(* Logix 5000 project; controller SX_V040001_C001 vendor 1 type 14 code 77 rev 16.23; software revision 16.04; part 24 of 35 *)
(* tags used below, declared in another part *)
   ALL_KINDS : INT[90];
   Basic : INT;
   DRIVE : INT[32];
   DRIVE_INTERVAL : INT[8];
   G_AInput : DINT[8];
   G_DInput : DINT[3];
   G_DOutput : DINT[3];
   Min_Counter : DINT;
   PARAMETER : INT[501];
(* MainProgram, continued *)

ROUTINE OperatingHours   (* ladder *)
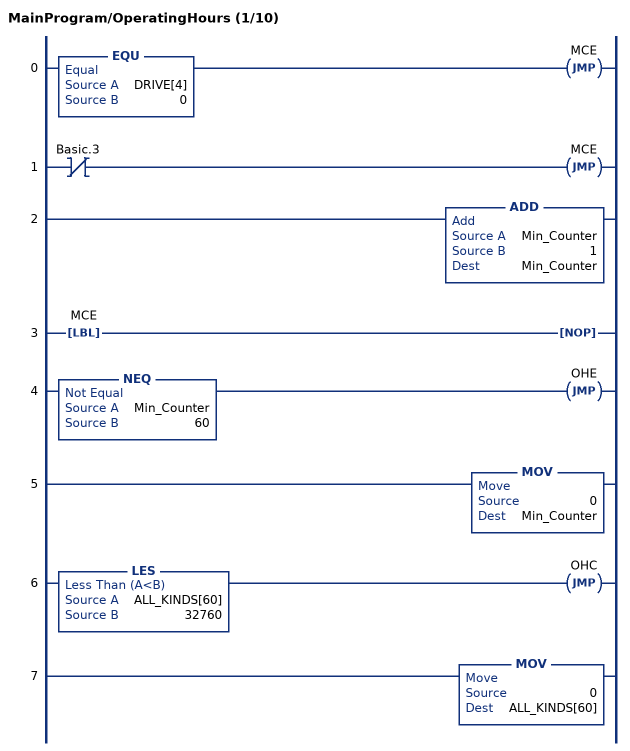
   0: EQU(DRIVE[4],0)JMP(MCE);
   1: XIO(Basic.3)JMP(MCE);
   2: ADD(Min_Counter,1,Min_Counter);
   3: LBL(MCE)NOP();
   4: NEQ(Min_Counter,60)JMP(OHE);
   5: MOV(0,Min_Counter);
   6: LES(ALL_KINDS[60],32760)JMP(OHC);
   7: MOV(0,ALL_KINDS[60]);
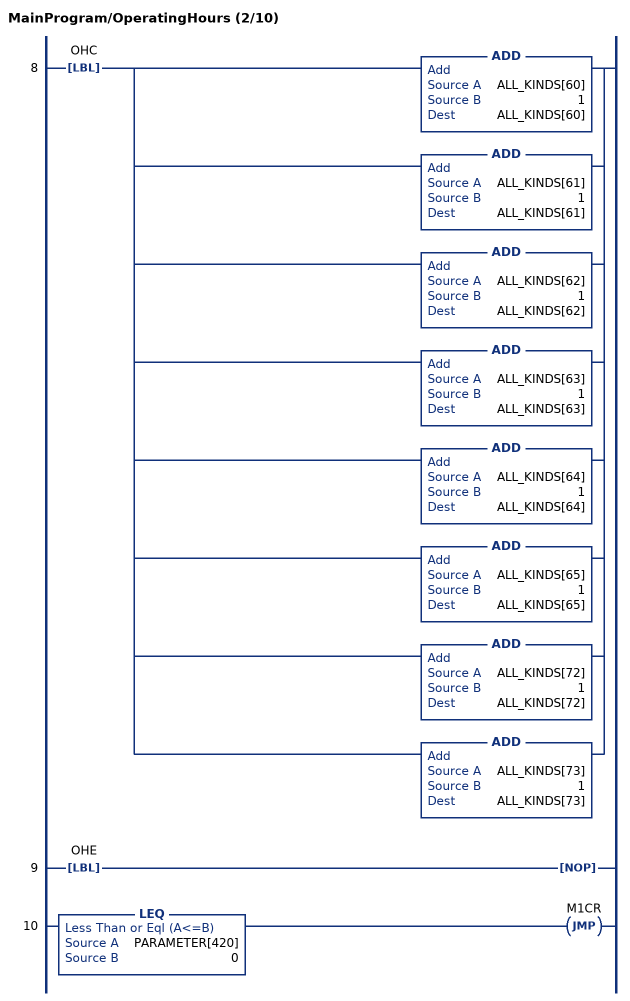
   8: LBL(OHC)[ADD(ALL_KINDS[60],1,ALL_KINDS[60]) ,ADD(ALL_KINDS[61],1,ALL_KINDS[61]) ,ADD(ALL_KINDS[62],1,ALL_KINDS[62]) ,ADD(ALL_KINDS[63],1,ALL_KINDS[63]) ,ADD(ALL_KINDS[64],1,ALL_KINDS[64]) ,ADD(ALL_KINDS[65],1,ALL_KINDS[65]) ,ADD(ALL_KINDS[72],1,ALL_KINDS[72]) ,ADD(ALL_KINDS[73],1,ALL_KINDS[73]) ];
   9: LBL(OHE)NOP();
   10: LEQ(PARAMETER[420],0)JMP(M1CR);
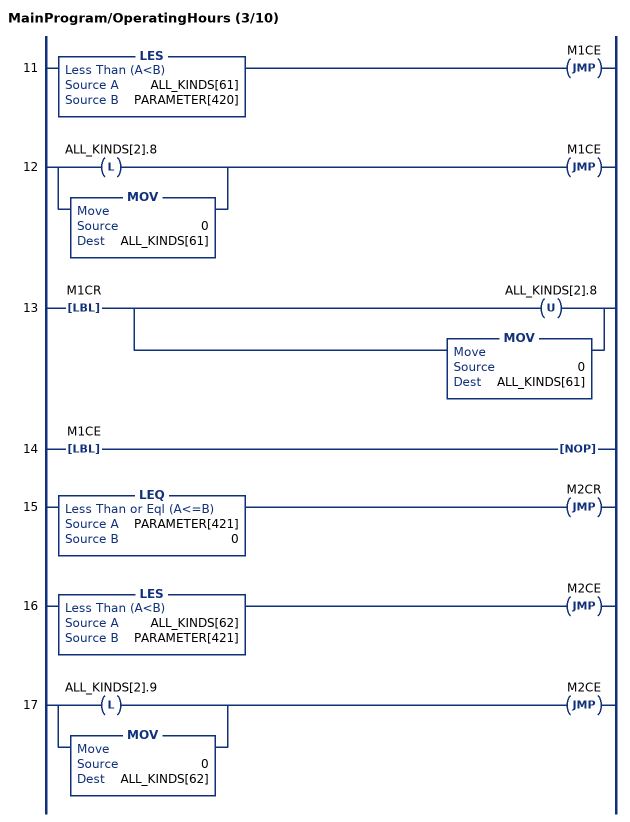
   11: LES(ALL_KINDS[61],PARAMETER[420])JMP(M1CE);
   12: [OTL(ALL_KINDS[2].8) ,MOV(0,ALL_KINDS[61]) ]JMP(M1CE);
   13: LBL(M1CR)[OTU(ALL_KINDS[2].8) ,MOV(0,ALL_KINDS[61]) ];
   14: LBL(M1CE)NOP();
   15: LEQ(PARAMETER[421],0)JMP(M2CR);
   16: LES(ALL_KINDS[62],PARAMETER[421])JMP(M2CE);
   17: [OTL(ALL_KINDS[2].9) ,MOV(0,ALL_KINDS[62]) ]JMP(M2CE);
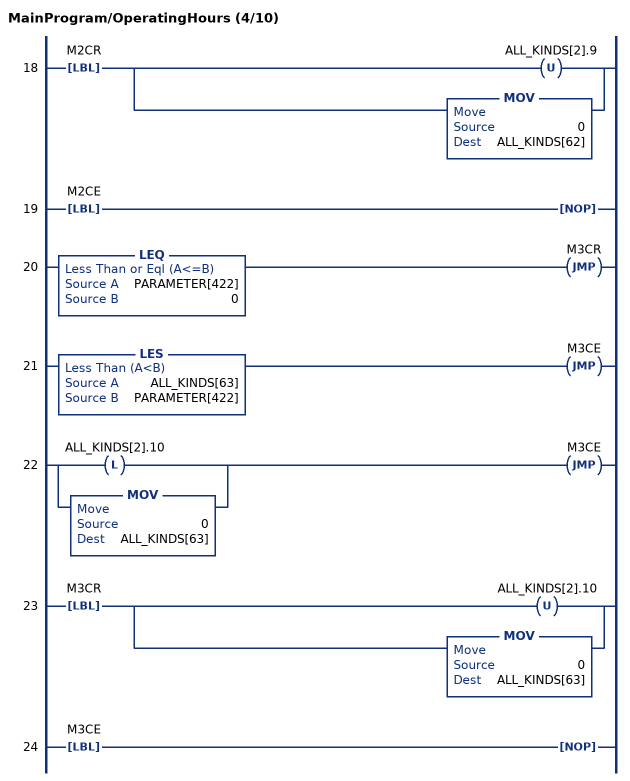
   18: LBL(M2CR)[OTU(ALL_KINDS[2].9) ,MOV(0,ALL_KINDS[62]) ];
   19: LBL(M2CE)NOP();
   20: LEQ(PARAMETER[422],0)JMP(M3CR);
   21: LES(ALL_KINDS[63],PARAMETER[422])JMP(M3CE);
   22: [OTL(ALL_KINDS[2].10) ,MOV(0,ALL_KINDS[63]) ]JMP(M3CE);
   23: LBL(M3CR)[OTU(ALL_KINDS[2].10) ,MOV(0,ALL_KINDS[63]) ];
   24: LBL(M3CE)NOP();
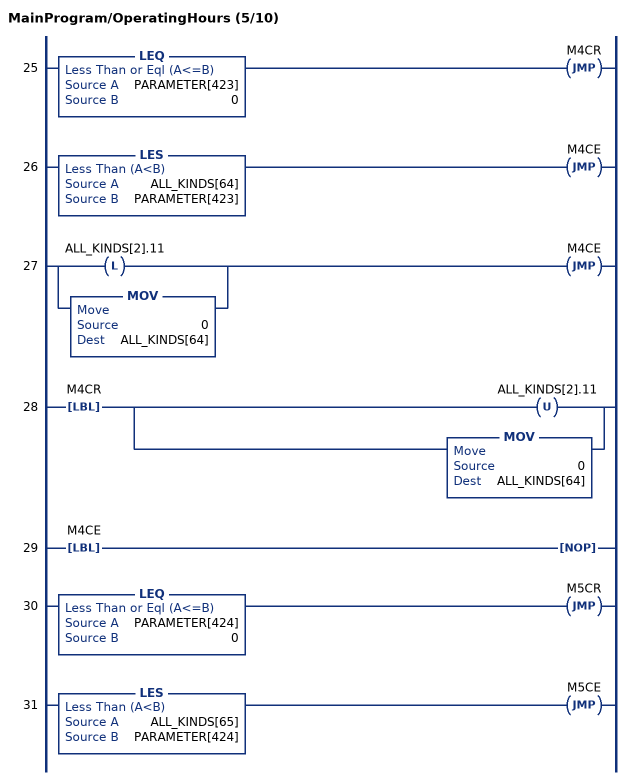
   25: LEQ(PARAMETER[423],0)JMP(M4CR);
   26: LES(ALL_KINDS[64],PARAMETER[423])JMP(M4CE);
   27: [OTL(ALL_KINDS[2].11) ,MOV(0,ALL_KINDS[64]) ]JMP(M4CE);
   28: LBL(M4CR)[OTU(ALL_KINDS[2].11) ,MOV(0,ALL_KINDS[64]) ];
   29: LBL(M4CE)NOP();
   30: LEQ(PARAMETER[424],0)JMP(M5CR);
   31: LES(ALL_KINDS[65],PARAMETER[424])JMP(M5CE);
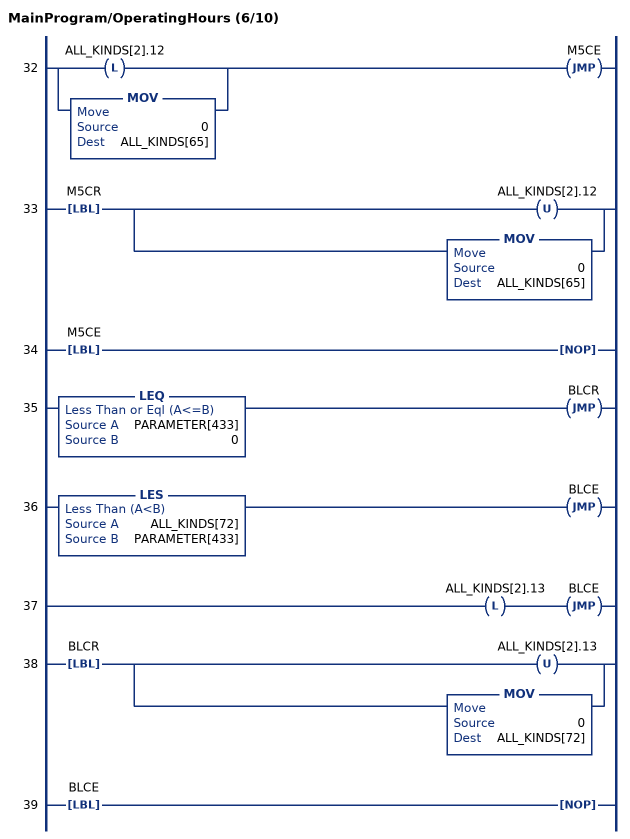
   32: [OTL(ALL_KINDS[2].12) ,MOV(0,ALL_KINDS[65]) ]JMP(M5CE);
   33: LBL(M5CR)[OTU(ALL_KINDS[2].12) ,MOV(0,ALL_KINDS[65]) ];
   34: LBL(M5CE)NOP();
   35: LEQ(PARAMETER[433],0)JMP(BLCR);
   36: LES(ALL_KINDS[72],PARAMETER[433])JMP(BLCE);
   37: OTL(ALL_KINDS[2].13)JMP(BLCE);
   38: LBL(BLCR)[OTU(ALL_KINDS[2].13) ,MOV(0,ALL_KINDS[72]) ];
   39: LBL(BLCE)NOP();
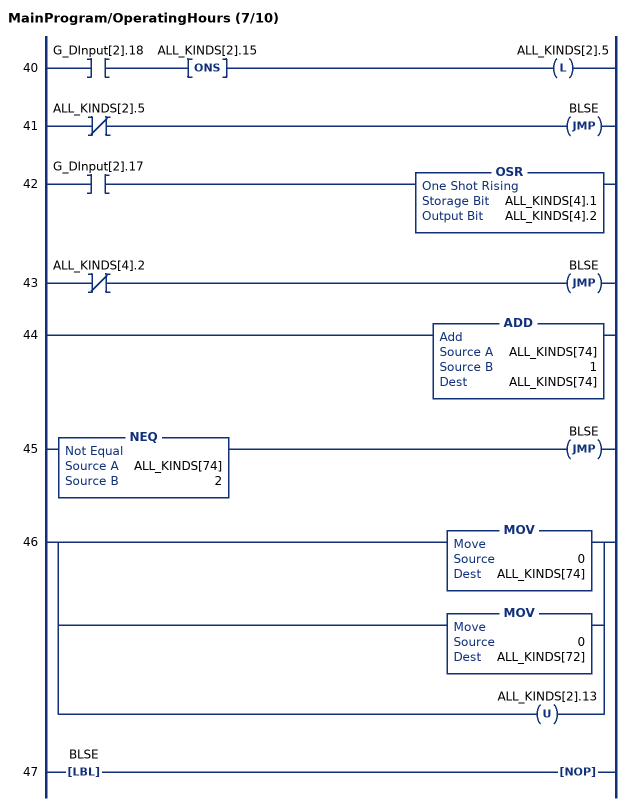
   40: XIC(G_DInput[2].18)ONS(ALL_KINDS[2].15)OTL(ALL_KINDS[2].5);
   41: XIO(ALL_KINDS[2].5)JMP(BLSE);
   42: XIC(G_DInput[2].17)OSR(ALL_KINDS[4].1,ALL_KINDS[4].2);
   43: XIO(ALL_KINDS[4].2)JMP(BLSE);
   44: ADD(ALL_KINDS[74],1,ALL_KINDS[74]);
   45: NEQ(ALL_KINDS[74],2)JMP(BLSE);
   46: [MOV(0,ALL_KINDS[74]) ,MOV(0,ALL_KINDS[72]) ,OTU(ALL_KINDS[2].13) ];
   47: LBL(BLSE)NOP();
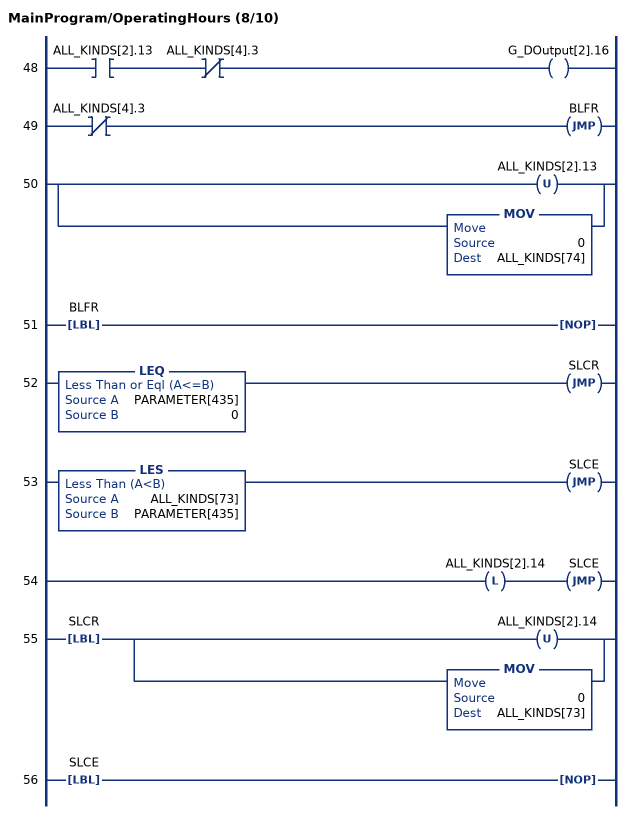
   48: XIC(ALL_KINDS[2].13)XIO(ALL_KINDS[4].3)OTE(G_DOutput[2].16);
   49: XIO(ALL_KINDS[4].3)JMP(BLFR);
   50: [OTU(ALL_KINDS[2].13) ,MOV(0,ALL_KINDS[74]) ];
   51: LBL(BLFR)NOP();
   52: LEQ(PARAMETER[435],0)JMP(SLCR);
   53: LES(ALL_KINDS[73],PARAMETER[435])JMP(SLCE);
   54: OTL(ALL_KINDS[2].14)JMP(SLCE);
   55: LBL(SLCR)[OTU(ALL_KINDS[2].14) ,MOV(0,ALL_KINDS[73]) ];
   56: LBL(SLCE)NOP();
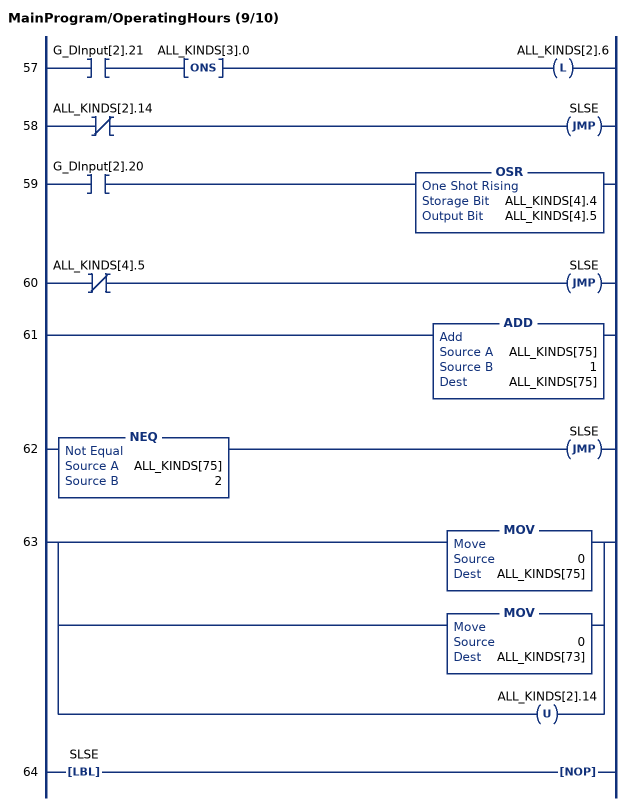
   57: XIC(G_DInput[2].21)ONS(ALL_KINDS[3].0)OTL(ALL_KINDS[2].6);
   58: XIO(ALL_KINDS[2].14)JMP(SLSE);
   59: XIC(G_DInput[2].20)OSR(ALL_KINDS[4].4,ALL_KINDS[4].5);
   60: XIO(ALL_KINDS[4].5)JMP(SLSE);
   61: ADD(ALL_KINDS[75],1,ALL_KINDS[75]);
   62: NEQ(ALL_KINDS[75],2)JMP(SLSE);
   63: [MOV(0,ALL_KINDS[75]) ,MOV(0,ALL_KINDS[73]) ,OTU(ALL_KINDS[2].14) ];
   64: LBL(SLSE)NOP();
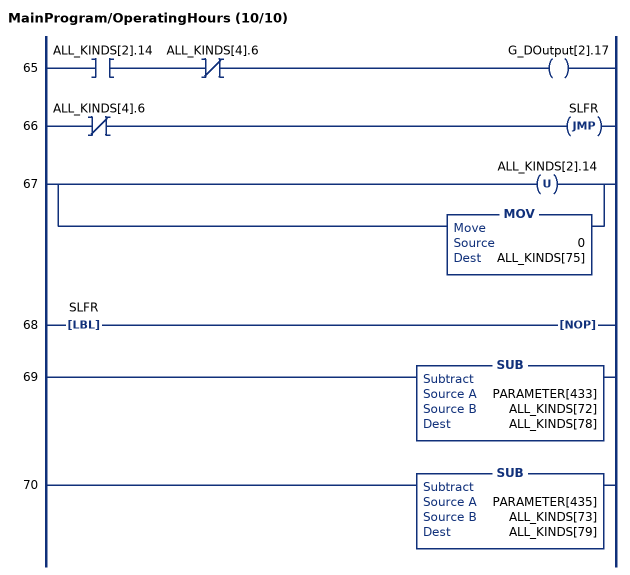
   65: XIC(ALL_KINDS[2].14)XIO(ALL_KINDS[4].6)OTE(G_DOutput[2].17);
   66: XIO(ALL_KINDS[4].6)JMP(SLFR);
   67: [OTU(ALL_KINDS[2].14) ,MOV(0,ALL_KINDS[75]) ];
   68: LBL(SLFR)NOP();
   69: SUB(PARAMETER[433],ALL_KINDS[72],ALL_KINDS[78]);
   70: SUB(PARAMETER[435],ALL_KINDS[73],ALL_KINDS[79]);
END_ROUTINE

ROUTINE ReadInput   (* ladder *)
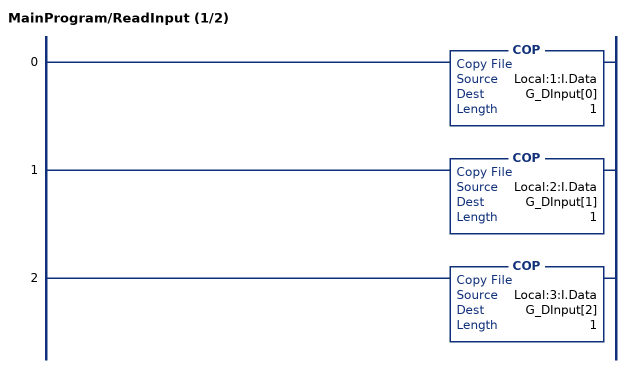
   0: COP(Local:1:I.Data,G_DInput[0],1);
   1: COP(Local:2:I.Data,G_DInput[1],1);
   2: COP(Local:3:I.Data,G_DInput[2],1);
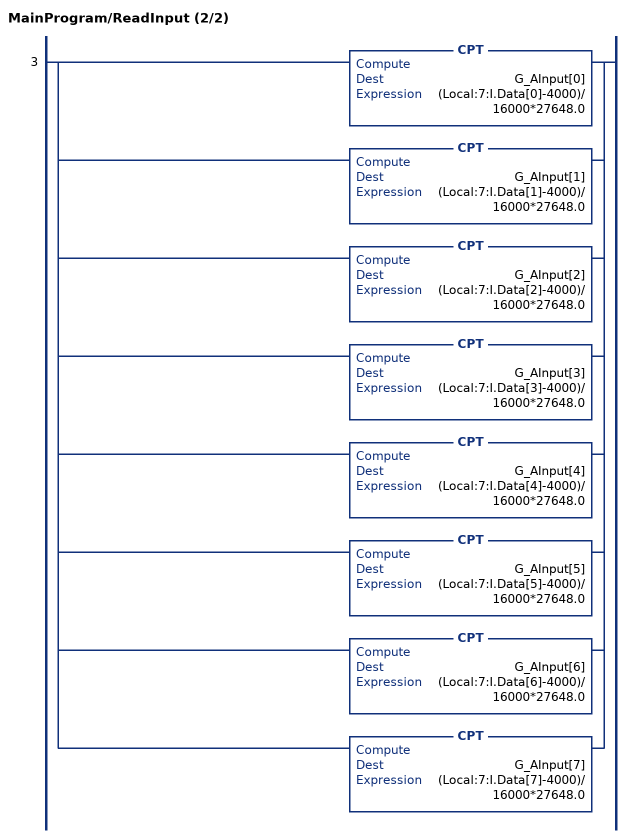
   3: [CPT(G_AInput[0],(Local:7:I.Data[0]-4000)/16000*27648.0) ,CPT(G_AInput[1],(Local:7:I.Data[1]-4000)/16000*27648.0) ,CPT(G_AInput[2],(Local:7:I.Data[2]-4000)/16000*27648.0) ,CPT(G_AInput[3],(Local:7:I.Data[3]-4000)/16000*27648.0) ,CPT(G_AInput[4],(Local:7:I.Data[4]-4000)/16000*27648.0) ,CPT(G_AInput[5],(Local:7:I.Data[5]-4000)/16000*27648.0) ,CPT(G_AInput[6],(Local:7:I.Data[6]-4000)/16000*27648.0) ,CPT(G_AInput[7],(Local:7:I.Data[7]-4000)/16000*27648.0) ];
END_ROUTINE

ROUTINE RecipeActions   (* ladder *)
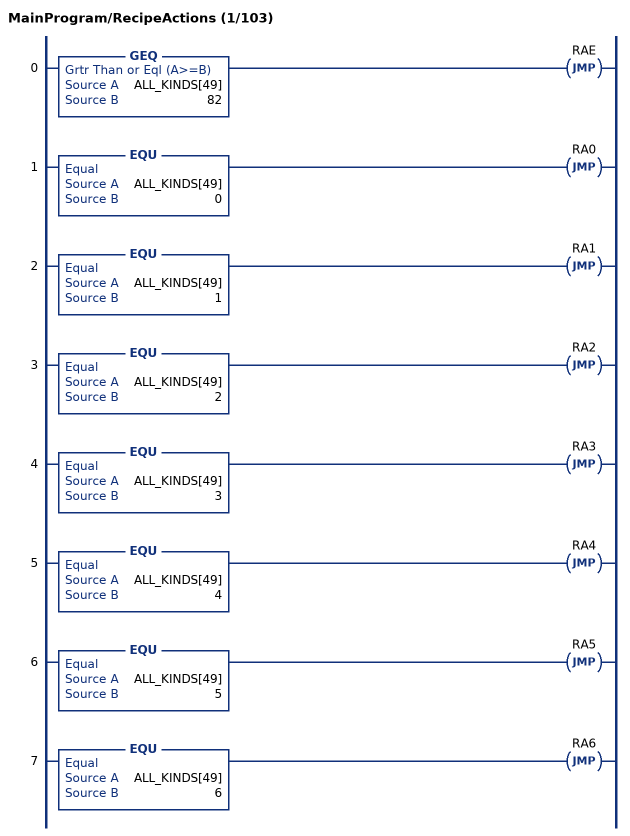
   0: GEQ(ALL_KINDS[49],82)JMP(RAE);
   1: EQU(ALL_KINDS[49],0)JMP(RA0);
   2: EQU(ALL_KINDS[49],1)JMP(RA1);
   3: EQU(ALL_KINDS[49],2)JMP(RA2);
   4: EQU(ALL_KINDS[49],3)JMP(RA3);
   5: EQU(ALL_KINDS[49],4)JMP(RA4);
   6: EQU(ALL_KINDS[49],5)JMP(RA5);
   7: EQU(ALL_KINDS[49],6)JMP(RA6);
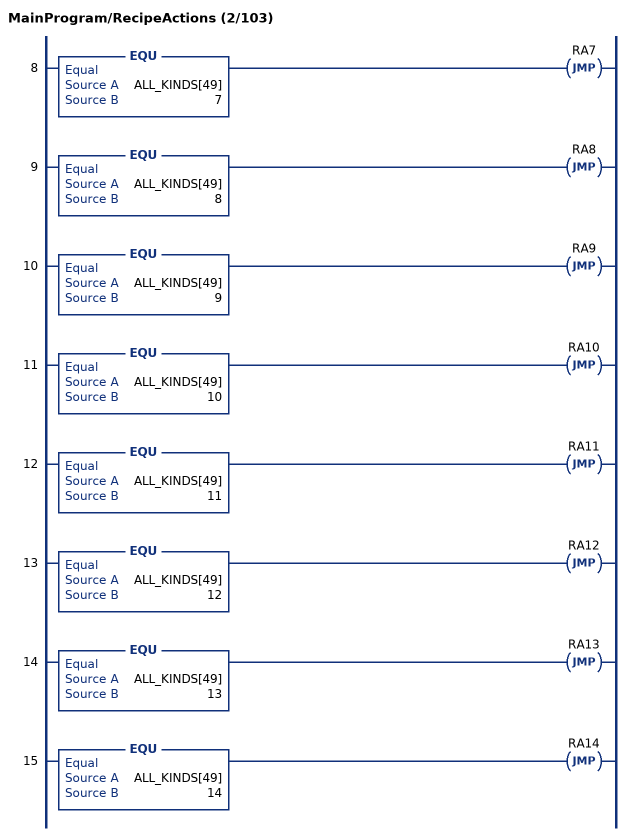
   8: EQU(ALL_KINDS[49],7)JMP(RA7);
   9: EQU(ALL_KINDS[49],8)JMP(RA8);
   10: EQU(ALL_KINDS[49],9)JMP(RA9);
   11: EQU(ALL_KINDS[49],10)JMP(RA10);
   12: EQU(ALL_KINDS[49],11)JMP(RA11);
   13: EQU(ALL_KINDS[49],12)JMP(RA12);
   14: EQU(ALL_KINDS[49],13)JMP(RA13);
   15: EQU(ALL_KINDS[49],14)JMP(RA14);
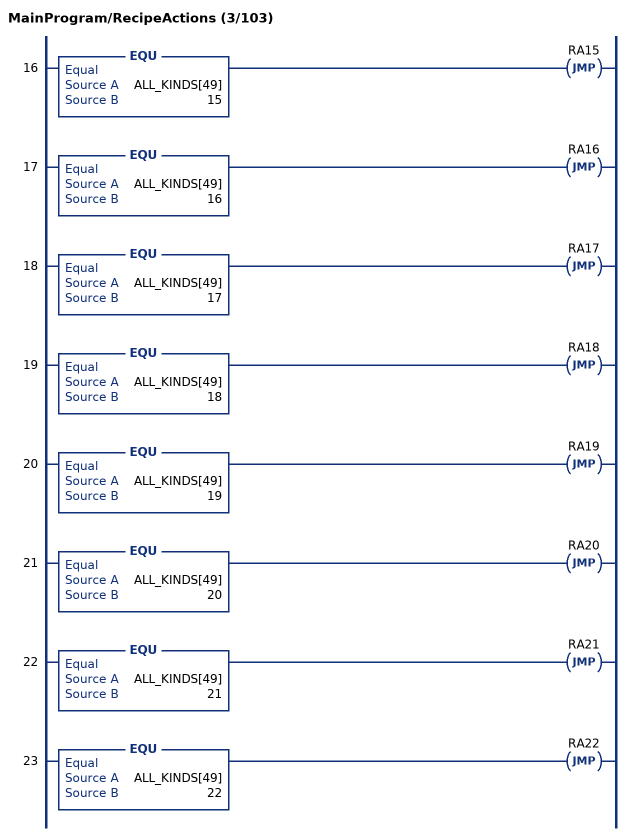
   16: EQU(ALL_KINDS[49],15)JMP(RA15);
   17: EQU(ALL_KINDS[49],16)JMP(RA16);
   18: EQU(ALL_KINDS[49],17)JMP(RA17);
   19: EQU(ALL_KINDS[49],18)JMP(RA18);
   20: EQU(ALL_KINDS[49],19)JMP(RA19);
   21: EQU(ALL_KINDS[49],20)JMP(RA20);
   22: EQU(ALL_KINDS[49],21)JMP(RA21);
   23: EQU(ALL_KINDS[49],22)JMP(RA22);
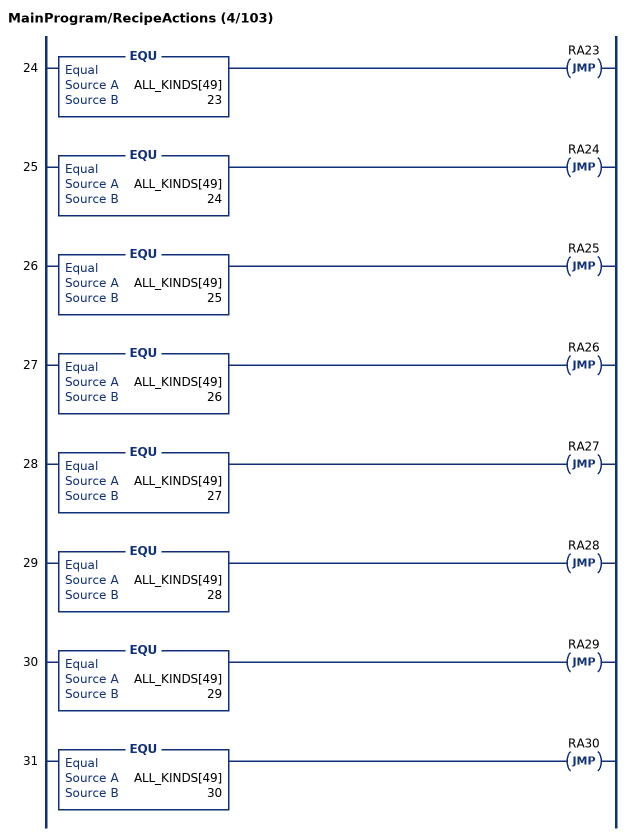
   24: EQU(ALL_KINDS[49],23)JMP(RA23);
   25: EQU(ALL_KINDS[49],24)JMP(RA24);
   26: EQU(ALL_KINDS[49],25)JMP(RA25);
   27: EQU(ALL_KINDS[49],26)JMP(RA26);
   28: EQU(ALL_KINDS[49],27)JMP(RA27);
   29: EQU(ALL_KINDS[49],28)JMP(RA28);
   30: EQU(ALL_KINDS[49],29)JMP(RA29);
   31: EQU(ALL_KINDS[49],30)JMP(RA30);
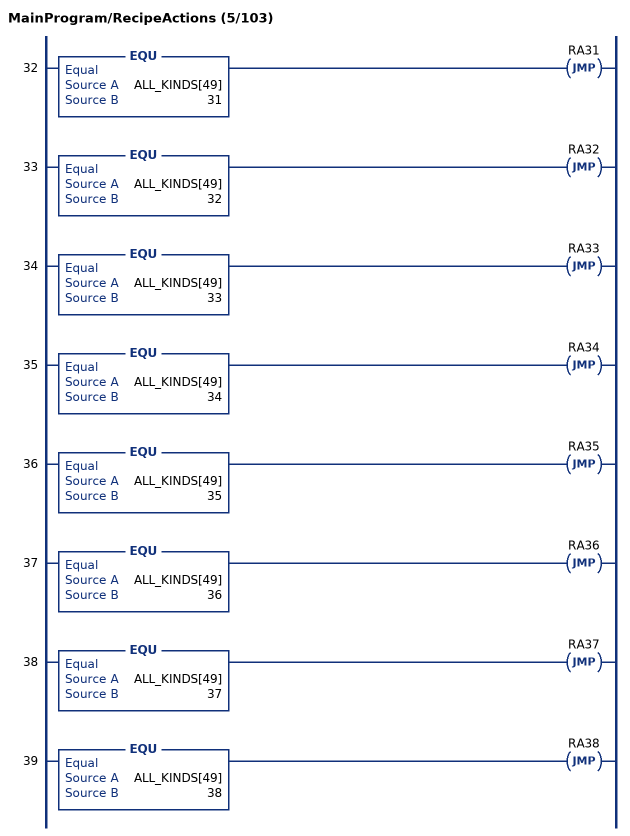
   32: EQU(ALL_KINDS[49],31)JMP(RA31);
   33: EQU(ALL_KINDS[49],32)JMP(RA32);
   34: EQU(ALL_KINDS[49],33)JMP(RA33);
   35: EQU(ALL_KINDS[49],34)JMP(RA34);
   36: EQU(ALL_KINDS[49],35)JMP(RA35);
   37: EQU(ALL_KINDS[49],36)JMP(RA36);
   38: EQU(ALL_KINDS[49],37)JMP(RA37);
   39: EQU(ALL_KINDS[49],38)JMP(RA38);
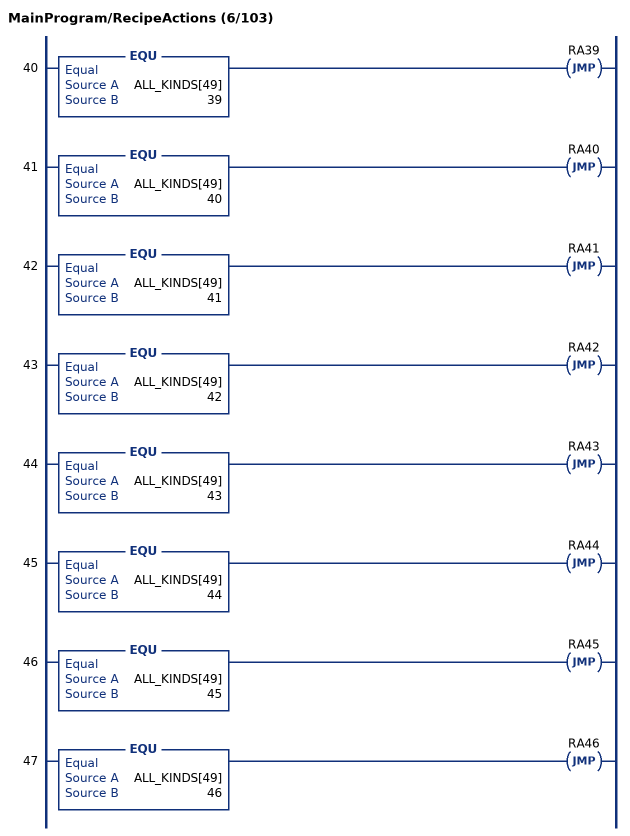
   40: EQU(ALL_KINDS[49],39)JMP(RA39);
   41: EQU(ALL_KINDS[49],40)JMP(RA40);
   42: EQU(ALL_KINDS[49],41)JMP(RA41);
   43: EQU(ALL_KINDS[49],42)JMP(RA42);
   44: EQU(ALL_KINDS[49],43)JMP(RA43);
   45: EQU(ALL_KINDS[49],44)JMP(RA44);
   46: EQU(ALL_KINDS[49],45)JMP(RA45);
   47: EQU(ALL_KINDS[49],46)JMP(RA46);
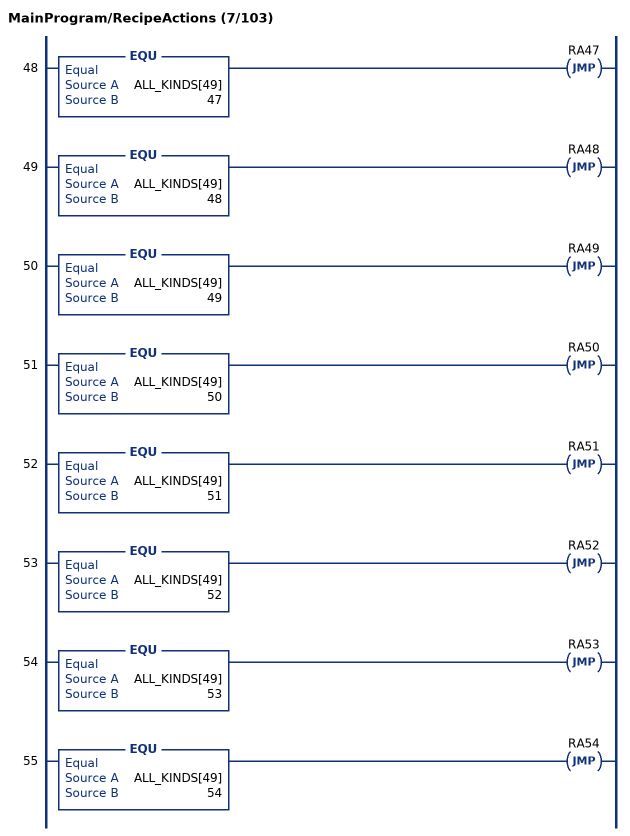
   48: EQU(ALL_KINDS[49],47)JMP(RA47);
   49: EQU(ALL_KINDS[49],48)JMP(RA48);
   50: EQU(ALL_KINDS[49],49)JMP(RA49);
   51: EQU(ALL_KINDS[49],50)JMP(RA50);
   52: EQU(ALL_KINDS[49],51)JMP(RA51);
   53: EQU(ALL_KINDS[49],52)JMP(RA52);
   54: EQU(ALL_KINDS[49],53)JMP(RA53);
   55: EQU(ALL_KINDS[49],54)JMP(RA54);
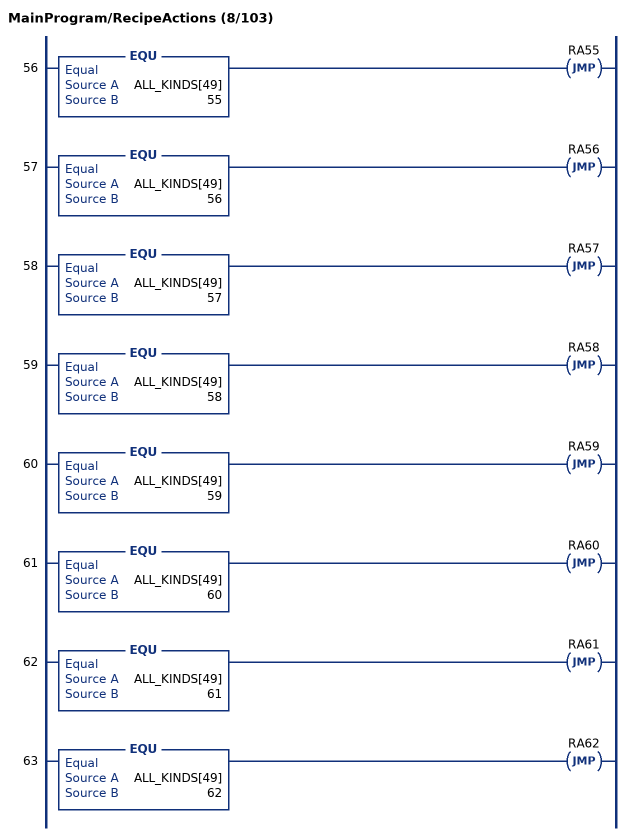
   56: EQU(ALL_KINDS[49],55)JMP(RA55);
   57: EQU(ALL_KINDS[49],56)JMP(RA56);
   58: EQU(ALL_KINDS[49],57)JMP(RA57);
   59: EQU(ALL_KINDS[49],58)JMP(RA58);
   60: EQU(ALL_KINDS[49],59)JMP(RA59);
   61: EQU(ALL_KINDS[49],60)JMP(RA60);
   62: EQU(ALL_KINDS[49],61)JMP(RA61);
   63: EQU(ALL_KINDS[49],62)JMP(RA62);
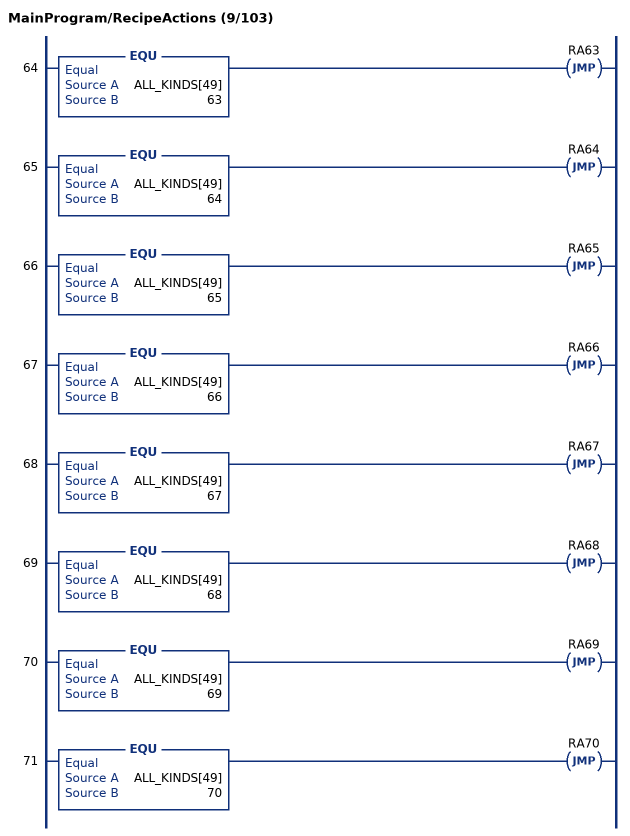
   64: EQU(ALL_KINDS[49],63)JMP(RA63);
   65: EQU(ALL_KINDS[49],64)JMP(RA64);
   66: EQU(ALL_KINDS[49],65)JMP(RA65);
   67: EQU(ALL_KINDS[49],66)JMP(RA66);
   68: EQU(ALL_KINDS[49],67)JMP(RA67);
   69: EQU(ALL_KINDS[49],68)JMP(RA68);
   70: EQU(ALL_KINDS[49],69)JMP(RA69);
   71: EQU(ALL_KINDS[49],70)JMP(RA70);
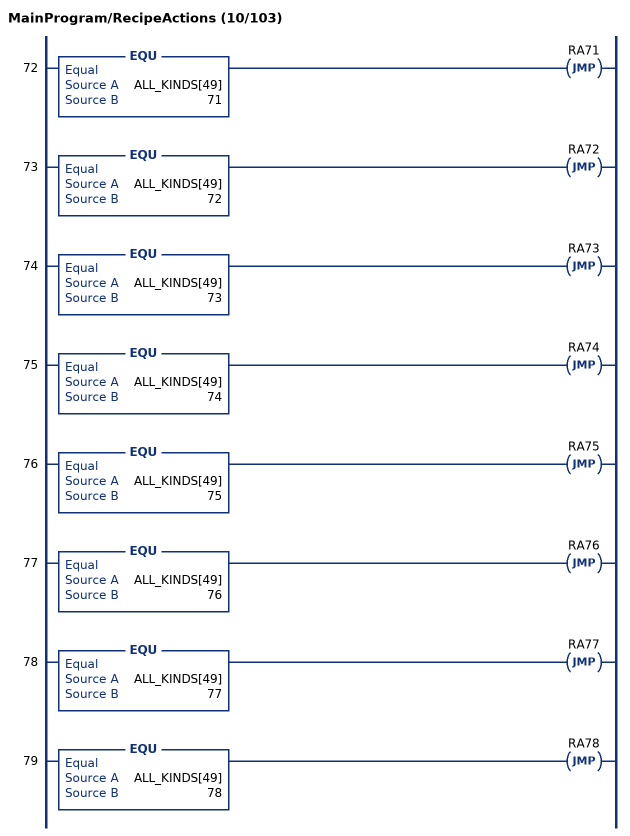
   72: EQU(ALL_KINDS[49],71)JMP(RA71);
   73: EQU(ALL_KINDS[49],72)JMP(RA72);
   74: EQU(ALL_KINDS[49],73)JMP(RA73);
   75: EQU(ALL_KINDS[49],74)JMP(RA74);
   76: EQU(ALL_KINDS[49],75)JMP(RA75);
   77: EQU(ALL_KINDS[49],76)JMP(RA76);
   78: EQU(ALL_KINDS[49],77)JMP(RA77);
   79: EQU(ALL_KINDS[49],78)JMP(RA78);
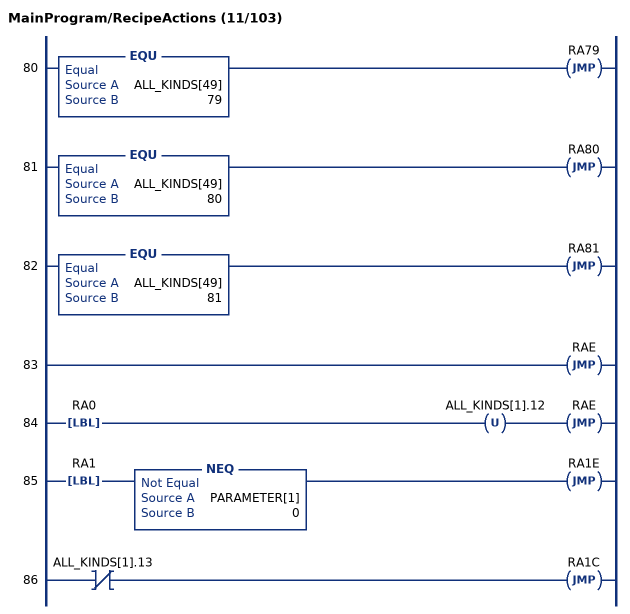
   80: EQU(ALL_KINDS[49],79)JMP(RA79);
   81: EQU(ALL_KINDS[49],80)JMP(RA80);
   82: EQU(ALL_KINDS[49],81)JMP(RA81);
   83: JMP(RAE);
   84: LBL(RA0)OTU(ALL_KINDS[1].12)JMP(RAE);
   85: LBL(RA1)NEQ(PARAMETER[1],0)JMP(RA1E);
   86: XIO(ALL_KINDS[1].13)JMP(RA1C);
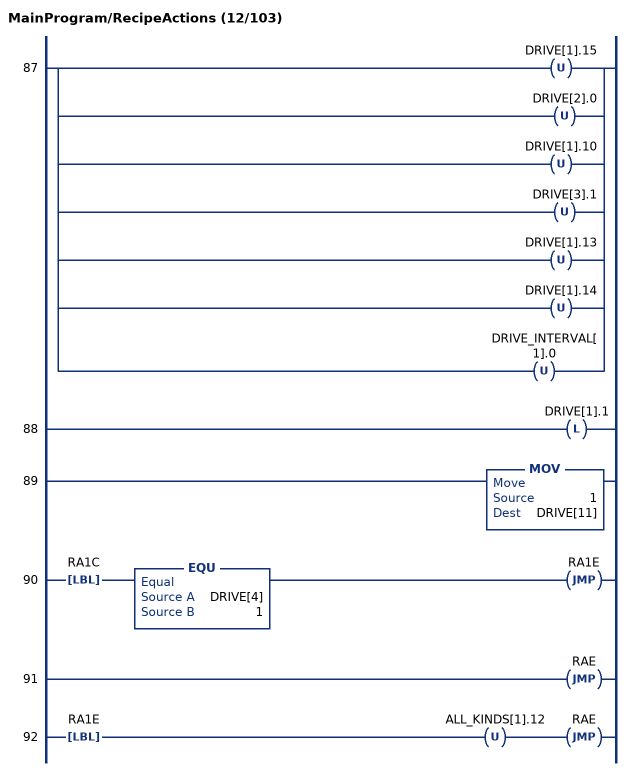
   87: [OTU(DRIVE[1].15) ,OTU(DRIVE[2].0) ,OTU(DRIVE[1].10) ,OTU(DRIVE[3].1) ,OTU(DRIVE[1].13) ,OTU(DRIVE[1].14) ,OTU(DRIVE_INTERVAL[1].0) ];
   88: OTL(DRIVE[1].1);
   89: MOV(1,DRIVE[11]);
   90: LBL(RA1C)EQU(DRIVE[4],1)JMP(RA1E);
   91: JMP(RAE);
   92: LBL(RA1E)OTU(ALL_KINDS[1].12)JMP(RAE);
